ABB RobotStudio station: Inverted.rspag

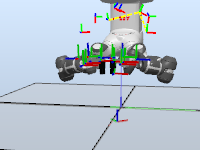
--- station ---
Station DEMO (saved by RobotStudio 20.4.9280.0)
Controller RW6.10.01
  mechanical unit ROB_R: IRB14000_0.5_0.5_R, 6 joints, base frame (0, 0, 820) mm, rotated rx 180 ry 0 rz 0 deg
  mechanical unit ROB_R_7: IRB14000_0.5_0.5_R, 1 joints, base frame (0, 0, 820) mm, rotated rx 180 ry 0 rz 0 deg
  mechanical unit ROB_L: IRB14000_0.5_0.5_L, 6 joints, base frame (0, 0, 820) mm, rotated rx 180 ry 0 rz 0 deg
  mechanical unit ROB_L_7: IRB14000_0.5_0.5_L, 1 joints, base frame (0, 0, 820) mm, rotated rx 180 ry 0 rz 0 deg
Layout (positions relative to the parent item):
  - IRB14000_0.5_0.5 [mechanism, from Robots\IRB14000_0.5_0.5__01.rslib] at (0, 0, 820) mm, rotated rx 180 ry 0 rz 0 deg
  - IRB14000_0.5_0.5_R [mechanism, from Robots\IRB14000_0.5_0.5__01.rslib] at (0, 0, 820) mm, rotated rx 180 ry 0 rz 0 deg; joint values [0.956, -0.6515, -0.6762, 0.5544, 3.1216, 1.0782, 0.2397] (rad or m)
  - IRB14000_0.5_0.5_L [mechanism, from Robots\IRB14000_0.5_0.5__01.rslib] at (0, 0, 820) mm, rotated rx 180 ry 0 rz 0 deg; joint values [-0.9175, -0.6335, 0.6594, 0.5525, 3.1588, 1.0767, -3.4124] (rad or m)
  - cam1 [part] at (530.01, -66.08, 390.5) mm, rotated rx -90 ry 1.82 rz -90 deg
  - cam2 [part] at (530.01, 64.49, 340.52) mm, rotated rx 90 ry 1.82 rz 90 deg
Attachment: cam2 is attached to IRB14000_0.5_0.5_R / Link7
Attachment: cam1 is attached to IRB14000_0.5_0.5_L / Link7
Targets, tools, work objects and paths stored in the station and not in the controller backup, written as RAPID:
! task T_ROB_R
MODULE MainModule
  VAR syncident synco;
  VAR syncident syncon;
  VAR syncident syncoff;
  VAR jointtarget jtraised10:=[[70.951,-118.367,40.9926,106.328,50.1338,-20.9947],[-83.9002,9E+09,9E+09,9E+09,9E+09,9E+09]];
  PROC runexperiment()
    Reset Collision_Avoidance;
    ConfL \Off;
    WaitSyncTask synco,tasklist;
    WaitTime nwaittime;
    WaitSyncTask synco,tasklist;
  ENDPROC
  PROC goto800()
    Reset Collision_Avoidance;
    ConfL \Off;
  ENDPROC
  PROC runallold()
    goto1100;
    goto1400;
    goto1100;
  ENDPROC
  PROC MainOld()
    Reset Collision_Avoidance;
  ENDPROC
  PROC Mainew()
    Reset Collision_Avoidance;
  ENDPROC
ENDMODULE

! task T_ROB_R
MODULE YuMiLib_Params_R
  TASK PERS tooldata tVacuum2:=[TRUE,[[-63.5,18.5,37.5],[0.707106781,0,-0.707106781,0]],[0.28,[7.1,11.9,47.3],[1,0,0,0],0.00025,0.00029,0.00012]];
  TASK PERS tooldata tVacuum1:=[TRUE,[[63.5,18.5,37.5],[0.707106781,0,0.707106781,0]],[0.248,[8.6,11.7,52.7],[1,0,0,0],0.00021,0.00024,0.00009]];
  TASK PERS tooldata tHandCamera:=[TRUE,[[-7.79332,26.2553,35.637],[0.507106,-0.492819,-0.512337,-0.487323]],[0.262,[7.8,11.9,50.7],[1,0,0,0],0.00022,0.00024,0.00009]];
  TASK PERS tooldata tGripper:=[TRUE,[[0,0,136],[1,0,0,0]],[0.23,[8.2,11.7,52],[1,0,0,0],0.00021,0.00024,0.00009]];
  TASK PERS wobjdata WObj_Vision:=[FALSE,TRUE,"",[[401.591,32.4092,0],[0.424655,-0.000000122,-0.000000191,0.905355]],[[0,0,0],[1,0,0,0]]];
  TASK PERS wobjdata WObj_FollowRobL:=[FALSE,FALSE,"ROB_L",[[0,0,0],[1,0,0,0]],[[0,0,0],[1,0,0,0]]];
ENDMODULE

! task T_ROB_R
MODULE YuMiLibExamplesR
  PERS wobjdata TrayWObj:=[FALSE,TRUE,"",[[0,0,0],[1,0,0,0]],[[0,0,0],[1,0,0,0]]];
  PROC YLExample_MoveYSyncProc()
    ConfL \Off;
    ConfL \On;
  ENDPROC
  PROC YLExample_MoveYCollision()
    ConfL \Off;
    ConfL \On;
  ENDPROC
ENDMODULE

! task T_ROB_R
MODULE Data
  TASK PERS tooldata tool1:=[TRUE,[[-49.461,-63.6951,27.321],[1,0,0,0]],[0.23,[-49.461,-63.6951,27.321],[1,0,0,0],0,0,0]];
  PERS tooldata tMarker:=[TRUE,[[0,0,14],[1,0,0,0]],[0.001,[0,0,0.001],[1,0,0,0],0,0,0]];
  TASK PERS tooldata camup:=[TRUE,[[-55.3,0,21.2],[1,0,0,0]],[0.23,[-55.3,0,21.2],[1,0,0,0],0,0,0]];
  PERS wobjdata woupsidedown:=[FALSE,TRUE,"",[[0,0,0],[1,0,0,0]],[[0,0,0],[1,0,0,0]]];
  PERS wobjdata wobj0New:=[FALSE,TRUE,"",[[0,0,0],[0,0,0,1]],[[0,0,0],[1,0,0,0]]];
  TASK PERS wobjdata flangeRobL:=[FALSE,FALSE,"ROB_L",[[0,0,0],[1,0,0,0]],[[0,0,0],[1,0,0,0]]];
  TASK PERS wobjdata flangeRobR:=[FALSE,FALSE,"ROB_R",[[0,0,0],[1,0,0,0]],[[0,0,0],[1,0,0,0]]];
  VAR syncident syncpoint;
  VAR syncident syncraise;
  VAR syncident syncbat1;
  VAR syncident syncbat2;
ENDMODULE

! task T_ROB_L
MODULE MainModule
  VAR syncident syncon;
  VAR syncident syncoff;
  PROC runexperiment()
    Reset Collision_Avoidance;
    ConfL \Off;
    WaitSyncTask synco,tasklist;
    WaitTime nwaittime;
    WaitSyncTask synco,tasklist;
  ENDPROC
  PROC goto800()
    Reset Collision_Avoidance;
    ConfL \Off;
  ENDPROC
  PROC runallold()
    goto1100;
    goto1400;
    goto1100;
  ENDPROC
ENDMODULE

! task T_ROB_L
MODULE YuMiLib_Params_L
  TASK PERS tooldata tVacuum2:=[TRUE,[[-63.5,18.5,37.5],[0.707106781,0,-0.707106781,0]],[0.28,[7.1,11.9,47.3],[1,0,0,0],0.00025,0.00029,0.00012]];
  TASK PERS tooldata tVacuum1:=[TRUE,[[63.5,18.5,37.5],[0.707106781,0,0.707106781,0]],[0.248,[8.6,11.7,52.7],[1,0,0,0],0.00021,0.00024,0.00009]];
  TASK PERS tooldata tHandCamera:=[TRUE,[[-7.79332,26.2553,35.637],[0.507106,-0.492819,-0.512337,-0.487323]],[0.262,[7.8,11.9,50.7],[1,0,0,0],0.00022,0.00024,0.00009]];
  TASK PERS tooldata tGripper:=[TRUE,[[0,0,136],[1,0,0,0]],[0.23,[8.2,11.7,52],[1,0,0,0],0.00021,0.00024,0.00009]];
  TASK PERS wobjdata WObj_Vision:=[FALSE,TRUE,"",[[401.591,32.4092,0],[0.424655,-0.000000122,-0.000000191,0.905355]],[[0,0,0],[1,0,0,0]]];
  TASK PERS wobjdata WObj_FollowRobR:=[FALSE,FALSE,"ROB_R",[[0,0,0],[1,0,0,0]],[[0,0,0],[1,0,0,0]]];
ENDMODULE

! task T_ROB_L
MODULE Data
  PERS tooldata tool1:=[TRUE,[[5.46165,-3.35898,214.586],[1,0,0,0]],[0.23,[0,0,0.001],[1,0,0,0],0,0,0]];
  TASK PERS tooldata camup:=[TRUE,[[55.3,0,21.2],[1,0,0,0]],[0.23,[-55.3,0,21.2],[1,0,0,0],0,0,0]];
  PERS wobjdata woupsidedown:=[FALSE,TRUE,"",[[0,0,-710],[0,0,0,1]],[[0,0,0],[1,0,0,0]]];
  TASK PERS wobjdata flangeRobL:=[FALSE,FALSE,"ROB_L",[[0,0,0],[1,0,0,0]],[[0,0,0],[1,0,0,0]]];
  TASK PERS wobjdata flangeRobR:=[FALSE,FALSE,"ROB_R",[[0,0,0],[1,0,0,0]],[[0,0,0],[1,0,0,0]]];
  PERS wobjdata floor:=[FALSE,TRUE,"",[[0,0,0],[1,0,0,0]],[[0,0,0],[1,0,0,0]]];
  PERS wobjdata basetest:=[FALSE,TRUE,"",[[0,0,410],[0,0,0,1]],[[0,0,0],[1,0,0,0]]];
  VAR syncident synco;
  VAR syncident syncraise;
  VAR syncident syncbat1;
  VAR syncident syncbat2;
  VAR syncident syncpoint;
ENDMODULE

! task T_ROB_L
MODULE YuMiLibExamplesL
  PERS wobjdata TrayWObj:=[FALSE,TRUE,"",[[0,0,0],[1,0,0,0]],[[0,0,0],[1,0,0,0]]];
  PROC YLExample_MoveYSyncProc()
    ConfL \Off;
    ConfL \On;
  ENDPROC
  PROC YLExample_MoveYCollision()
    ConfL \Off;
    ConfL \On;
  ENDPROC
ENDMODULE


--- Backups/RW6.10.01/RAPID/TASK1/PROGMOD/Data.mod ---
MODULE Data

    ! Tooldata for the right camera.
    TASK PERS tooldata tCamR:=[TRUE,[[-55.3,0,21.2],[1,0,0,0]],[0.23,[-55.3,0,21.2],[1,0,0,0],0,0,0]];
    TASK PERS tooldata tCamR_orig:=[TRUE,[[-55.3,0,21.2],[1,0,0,0]],[0.23,[-55.3,0,21.2],[1,0,0,0],0,0,0]];

    TASK PERS robtarget origR := [[456,35,1099.44],[0.507892,0.491981,0.507892,0.491981],[1,2,0,4],[165,9E+9,9E+9,9E+9,9E+9,9E+9]];
    !Additional rotational adjustments

    !Additional rotational adjustments
    VAR num x_offs:=0.0;
    VAR num y_offs:=0;!0.12;
    VAR num z_offs:=0;!-1.00;

    !Data for the experiment
    VAR num distances{20}:=[50,60,70,80,90,100,110,120,130,140,150,160,170,180,190,200,210,220,230,240];
    PERS num nWaittime:=5;
    PERS wobjdata wobjHeart:=[FALSE,TRUE,"",[[0,0,1550],[0,0,1,0]],[[0,0,0],[1,0,0,0]]];
    PERS speeddata speedSlow:=[50,50,5000,5000];
    PERS num nRadius{2}:=[1100, 1400];
    PERS pos convergencePos{2} := [[0, 0, 0], [0, 0, 300]]; !z will be added to this position!

    !Adjusting the x and z position of the convergence points.
    PERS num x:= 456;
    PERS num z:= 1550;



    !For synchronization
    PERS tasks tasklist{2}:=[["T_ROB_R"],["T_ROB_L"]];
    VAR syncident syncpoint;

    !The Stereo2 app reads this status message and displays it on the Flexpendant.
    PERS string myStatus:="Dist 110 h = 1100";


    !For moving into a raised position and to resting aka 'bat' position
    VAR syncident syncraise;
    VAR syncident syncbat1;
    VAR syncident syncbat2;
    VAR jointtarget jtraised:=[[66.0331,-85.1911,41.3253,139.052,44.5799,5.71225],[-62.1903,9E+09,9E+09,9E+09,9E+09,9E+09]];
    VAR jointtarget jtbat:=[[64.6304,-143.384,34.5095,60.7933,53.7269,8.84934],[-140.721,9E+09,9E+09,9E+09,9E+09,9E+09]];
    VAR jointtarget jtraisedVia:=[[70.951,-118.367,40.9926,106.328,50.1338,-20.9947],[-83.9002,9E+09,9E+09,9E+09,9E+09,9E+09]];


ENDMODULE

--- Backups/RW6.10.01/RAPID/TASK1/PROGMOD/MainModule.mod ---
MODULE MainModule




    PROC Main()
        runall;
    ENDPROC

    PROC goToCalibPos()
        VAR jointtarget calibPos := [[-0.00840108,-129.997,30.0284,-0.019315,40.0852,-0.0138285],[-135.001,9E+09,9E+09,9E+09,9E+09,9E+09]];
        MoveAbsJ calibPos\NoEOffs,v1000,z50,tool0;
    ENDPROC

    PROC runall()

        FOR i FROM 1 TO DIM(nRadius, 1) DO
            runtest convergencePos{i}, nRadius{i};
        ENDFOR
    ENDPROC



    PROC MoveToDist(num dist,num h\speeddata sp, PERS wobjdata wobjHeart)
        VAR robtarget position:=[[365,-10,1000],[0.5,0.5,0.5,0.5],[1,-2,-2,4],[165,9E+09,9E+09,9E+09,9E+09,9E+09]];
        VAR num angle;
        VAR num halfdist;
        VAR num rads;
        VAR num zh;
        VAR num y;
        VAR speeddata speed;


        halfdist:=dist/2;
        speed:=speedSlow;
        angle:=ASin(halfdist/h);
        y:=h*sin(angle);
        zh:=h*cos(angle);

        position.trans:=[x,y,zh];
        IF Present(sp) THEN
            speed:=sp;
        ENDIF

        MoveL RelTool(position,0,0,0\Rx:=x_offs\Ry:=y_offs\Rz:=-(angle+z_offs)),speed,fine,tCamR\WObj:=wobjHeart;

    ENDPROC


    PROC inc()
        VAR num s:=1;
        z := z + s;
        goto1100;
    ENDPROC


    PROC incinc()

        VAR num s:=5;
        z := z + s;
        goto1100;
    ENDPROC


    PROC dec()

        VAR num s:=-1;
        z := z + s;
        goto1100;
    ENDPROC


    PROC decdec()
        VAR num s:=-5;
        z := z + s;
        goto1100;
    ENDPROC

    PROC incX()
        VAR num s:=1;
        x:=x+s;
        goto1100;
    ENDPROC


    PROC incincX()

        VAR num s:=5;
        x:=x+s;
        goto1100;
    ENDPROC


    PROC decX()

        VAR num s:=-1;
        x:=x+s;
        goto1100;
    ENDPROC


    PROC decdecX()

        VAR num s:=-5;
        x:=x+s;
        goto1100;
    ENDPROC

    PROC gotoX1()
        ReSet Collision_Avoidance;
        ConfL\Off;
        wobjHeart.uframe.trans := [convergencePos{1}.x, convergencePos{1}.y, convergencePos{1}.z + z];
        WaitSyncTask syncpoint,tasklist;
        !origR := CRobT(\Tool:=tCamR_orig);
        MoveToDist distances{3},nRadius{1}\sp:=v100, wobjHeart;
    ENDPROC

    PROC L_update()

    ENDPROC


    PROC R_update()
        VAR robtarget new;
        VAR pose orig_pose;
        VAR pose new_pose;
        VAR pose diff;
        VAR pose tool_pose;
        VAR btnres answer;
        tool_pose := tCamR_orig.tframe;
        new := CRobT(\Tool:=tCamR_orig);
        orig_pose := [origR.trans, origR.rot];
        new_pose := [new.trans, new.rot];
        diff := PoseMult(PoseInv(new_pose), orig_pose);
        tCamR.tframe := PoseMult(tool_pose, diff);


    ENDPROC

    PROC reset_tool()
        tCamR := tCamR_orig;

    ENDPROC

    PROC gotoX2()

        ReSet Collision_Avoidance;
        ConfL\Off;
        wobjHeart.uframe.trans := [convergencePos{1}.x, convergencePos{1}.y, convergencePos{1}.z+z];
        WaitSyncTask syncpoint,tasklist;
        MoveToDist distances{15},nRadius{1}\sp:=v100, wobjHeart;

    ENDPROC


    PROC gofrombatpos()

        ReSet Collision_Avoidance;
        ConfL\Off;
        MoveAbsJ jtraisedVia\NoEOffs,v100,fine,tCamR;
        MoveAbsJ jtraised\NoEOffs,v100,fine,tCamR;
        WaitSyncTask syncraise,tasklist;
    ENDPROC

    PROC gotoraisedpos()
        ReSet Collision_Avoidance;
        ConfL\Off;
        MoveAbsJ jtraised\NoEOffs,v100,fine,tCamR;
        WaitSyncTask syncraise,tasklist;

    ENDPROC

    PROC gotobatpos()
        ReSet Collision_Avoidance;
        ConfL\Off;
        MoveAbsJ jtraised\NoEOffs,v100,fine,tCamR\WObj:=wobjHeart;
        WaitSyncTask syncbat1,tasklist;
        WaitSyncTask syncbat2,tasklist;
        MoveAbsJ jtraisedVia\NoEOffs,v100,fine,tCamR;
        MoveAbsJ jtbat\NoEOffs,v100,fine,tCamR;

    ENDPROC



    PROC goto1100()
        ReSet Collision_Avoidance;
        ConfL\Off;
        wobjHeart.uframe.trans := [convergencePos{1}.x, convergencePos{1}.y, convergencePos{1}.z + z];
        WaitSyncTask syncpoint,tasklist;
        MoveToDist distances{1},nRadius{1}\sp:=v100, wobjHeart;
    ENDPROC


    PROC goto1400()
        ReSet Collision_Avoidance;
        ConfL\Off;
        wobjHeart.uframe.trans := [convergencePos{2}.x, convergencePos{2}.y, convergencePos{2}.z + z];
        WaitSyncTask syncpoint,tasklist;
        MoveToDist distances{1},nRadius{2}\sp:=v100, wobjHeart;

    ENDPROC


    PROC run1100()
        runtest convergencePos{1},nRadius{1};
    ENDPROC

    PROC run1400()

        runtest convergencePos{2},nRadius{2};
    ENDPROC



    PROC runtest(pos position,num h)

        ConfL\Off;
        wobjHeart.uframe.trans:=[position.x, position.y, position.z + z];
        WaitSyncTask syncpoint,tasklist;
        ReSet Collision_Avoidance;
        MoveToDist distances{1},h\sp:=v100, wobjHeart;

        FOR i FROM 1 TO Dim(distances,1) DO

            WaitSyncTask syncpoint,tasklist;
            myStatus:="Dist "+NumToStr(distances{i},0)+" h = "+NumToStr(h,0);
            ErrWrite\I,"Started moving. Dist "+NumToStr(distances{i},0)+" h = "+NumToStr(h,0),"";
            MoveToDist distances{i},h, wobjHeart;
            WaitTime nwaittime;
        ENDFOR
        WaitSyncTask syncpoint,tasklist;
    ENDPROC


ENDMODULE

--- Backups/RW6.10.01/RAPID/TASK2/PROGMOD/Data.mod ---
    MODULE Data


    ! Tooldata for the left camera.
    TASK PERS tooldata tCamL:=[TRUE,[[55.3,0,21.2],[1,0,0,0]],[0.23,[55.3,0,21.2],[1,0,0,0],0,0,0]];
    TASK PERS tooldata tCamL_orig:=[TRUE,[[55.3,0,21.2],[1,0,0,0]],[0.23,[55.3,0,21.2],[1,0,0,0],0,0,0]];

    TASK PERS robtarget origL := [[456,-35,1099.44],[0.491981,0.507892,0.491981,0.507892],[-1,2,-2,4],[-163.142,9E+9,9E+9,9E+9,9E+9,9E+9]];

   ! Additional rotational adjustments.
    VAR num x_offs:= 0.0;
    VAR num y_offs:= 0.0;
    VAR num z_offs:=0;!0.43;


    !Data for the experiment. These are shared with the right task and assigned in T_ROB_R/Data
    VAR num distances{20}:=[50,60,70,80,90,100,110,120,130,140,150,160,170,180,190,200,210,220,230,240];
    PERS num nWaittime;
    PERS wobjdata wobjHeart;
    PERS speeddata speedSlow;
    PERS num nRadius{2};
    PERS pos convergencePos{2};


    !Adjusting the x and z position of the convergence points.
    PERS num x;
    PERS num z;



    !For synchronization
    PERS tasks tasklist{2}:=[["T_ROB_R"],["T_ROB_L"]];
    VAR syncident syncpoint;

    !For moving into a raised position and to resting aka 'bat' position
    VAR jointtarget jtraised:=[[-74.7004,-91.3236,43.3868,218.306,45.6835,-171.438],[61.909,9E+09,9E+09,9E+09,9E+09,9E+09]];
    VAR syncident syncraise;
    VAR syncident syncbat1;
    VAR syncident syncbat2;
    VAR jointtarget jtbat:=[[-56.5752,-119.517,21.4015,271.499,49.3732,-213.567],[155.307,9E+09,9E+09,9E+09,9E+09,9E+09]];

ENDMODULE

--- Backups/RW6.10.01/RAPID/TASK2/PROGMOD/MainModule.mod ---
    MODULE MainModule



    PROC goToCalibPos()
        VAR jointtarget calibPos := [[0.00341333,-129.995,30.0196,-0.000788279,40.0913,-0.461743],[134.997,9E+09,9E+09,9E+09,9E+09,9E+09]];
        MoveAbsJ calibPos\NoEOffs,v1000,z50,tool0;
    ENDPROC

    PROC Main()

        runall;
    ENDPROC

    PROC runall()
        FOR i FROM 1 TO DIM(nRadius, 1) DO
            runtest convergencePos{i}, nRadius{i};
        ENDFOR
    ENDPROC



    PROC MoveToDist(num dist,num h,\speeddata sp, PERS wobjdata wobjHeart)
        !   VAR robtarget position := [[0,0,0],[0.0,0.0,0.7071,-0.7071],[1,1,0,4],[143.284,9E+09,9E+09,9E+09,9E+09,9E+09]];
        VAR robtarget position:=[[0,0,0],[0.5,0.5,0.5,0.5],[1,-2,0,0],[-163.142,9E+09,9E+09,9E+09,9E+09,9E+09]];
        VAR num angle;
        VAR num halfdist;
        VAR num rads;
        VAR num zh;
        VAR num y;
        VAR speeddata speed;

        halfdist:=dist/2;
        speed:=speedSlow;
        angle:=ASin(halfdist/h);
        y:=h*sin(angle);
        zh:=h*cos(angle);

        position.trans:=[x,-y,zh];
        IF Present(sp) THEN
            speed:=sp;
        ENDIF
        MoveL RelTool(position,0,0,0\Ry:=y_offs\Rz:=angle+z_offs),speed,fine,tCamL\WObj:=wobjHeart;


    ENDPROC





    PROC gotoraisedpos()

        ReSet Collision_Avoidance;
        ConfL\Off;
        WaitSyncTask syncraise,tasklist;
        MoveAbsJ jtraised\NoEOffs,v100,fine,tCamL;

    ENDPROC

    PROC inc()
        goto1100;
    ENDPROC


    PROC incinc()
        goto1100;
    ENDPROC


    PROC dec()
        goto1100;
    ENDPROC


    PROC decdec()
        goto1100;
    ENDPROC



    PROC incX()
        goto1100;
    ENDPROC


    PROC incincX()

        goto1100;
    ENDPROC


    PROC decX()

        goto1100;

    ENDPROC


    PROC decdecX()
        goto1100;

    ENDPROC

    PROC gofrombatpos()
        VAR jointtarget jtVia := [[-68.4054,-105.589,37.6928,245.742,40.601,-189.436],[135.726,9E+09,9E+09,9E+09,9E+09,9E+09]];
        ReSet Collision_Avoidance;
        ConfL\Off;
        WaitSyncTask syncraise,tasklist;
        MoveAbsJ jtVia\NoEOffs,v100,fine,tCamL;
        MoveAbsJ jtraised\NoEOffs,v100,fine,tCamL;

    ENDPROC

    PROC gotobatpos()
        VAR jointtarget jtBatPos := [[-68.4054,-105.589,37.6928,245.742,40.601,-189.436],[135.726,9E+09,9E+09,9E+09,9E+09,9E+09]];
        ReSet Collision_Avoidance;
        ConfL\Off;
        MoveAbsJ jtraised\NoEOffs,v100,fine,tCamL;
        WaitSyncTask syncbat1,tasklist;
        MoveAbsJ jtBatPos\NoEOffs,v100,fine,tCamL;
        MoveAbsJ jtbat\NoEOffs,v100,fine,tCamL;
        WaitSyncTask syncbat2,tasklist;
    ENDPROC


    PROC gotoX1()

        ReSet Collision_Avoidance;
        ConfL\Off;
        WaitSyncTask syncpoint,tasklist;
        !origL := CRobT(\Tool:=tCamL_orig);

        MoveToDist distances{3},nRadius{1}\sp:=v100, wobjHeart;
    ENDPROC


    PROC L_update()
        VAR robtarget new;
        VAR pose orig_pose;
        VAR pose new_pose;
        VAR pose diff;
        VAR pose tool_pose;
        VAR btnres answer;
        tool_pose := tCamL_orig.tframe;
        new := CRobT(\Tool:=tCamL_orig);
        orig_pose := [origL.trans, origL.rot];
        new_pose := [new.trans, new.rot];
        diff := PoseMult(PoseInv(new_pose), orig_pose);
        tCamL.tframe := PoseMult(tool_pose, diff);


    ENDPROC


    PROC R_update()
    ENDPROC

    PROC reset_tool()
        tCamL := tCamL_orig;

    ENDPROC

    PROC gotoX2()
        ReSet Collision_Avoidance;
        ConfL\Off;
        WaitSyncTask syncpoint,tasklist;
        MoveToDist distances{15},nRadius{1}\sp:=v100, wobjHeart;

    ENDPROC


    PROC goto1100()
        ReSet Collision_Avoidance;
        ConfL\Off;
        WaitSyncTask syncpoint,tasklist;
        MoveToDist distances{1},nRadius{1}\sp:=v100, wobjHeart;

    ENDPROC




    PROC goto1400()
        ReSet Collision_Avoidance;
        ConfL\Off;
        WaitSyncTask syncpoint,tasklist;
        MoveToDist distances{1},nRadius{2}\sp:=v100, wobjHeart;

    ENDPROC


    PROC run1100()
        runtest convergencePos{1},nRadius{1};
    ENDPROC

    PROC run1400()

        runtest convergencePos{2},nRadius{2};
    ENDPROC



    PROC runtest(pos position,num h)
        ReSet Collision_Avoidance;
        ConfL\Off;
        WaitSyncTask syncpoint,tasklist;

        MoveToDist distances{1},h\sp:=v100, wobjHeart;

        FOR i FROM 1 TO Dim(distances,1) DO
            WaitSyncTask syncpoint,tasklist;
            MoveToDist distances{i},h, wobjHeart;
            WaitTime nwaittime;
        ENDFOR

        WaitSyncTask syncpoint,tasklist;
    ENDPROC

ENDMODULE

--- Backups/RW6.10.01/SYSPAR/EIO.cfg ---
EIO:CFG_1.0:6:1::
#
SYSSIG_IN:

      -Signal "Collision_Avoidance" -Action "CollAvoidance"
#
INDUSTRIAL_NETWORK:

      -Name "DeviceNet" -Label "DeviceNet Master/Slave Network" -Address "2"
#
EIO_CROSS:

      -Name "Cross_Signal_Lamp" -Res "Signal_Lamp" -Act1 "DRV1BRAKE"
#
EIO_SIGNAL_SAFELEVEL:

      -Name "FlangePowerSafeLevel" -ActionWhenStartup "Last"

      -Name "SGcmdSafeLevel" -ActionWhenAccessible "Default"
#
ETHERNETIP_DEVICE:

      -Name "Hand_R" -StateWhenStartup "Deactivated" -VendorName "ABB"\
      -ProductName "EtherNet/IP EIP" -Label "2" -Address "192.168.125.30"\
      -VendorId 75 -ProductCode 1 -OutputAssembly 100 -InputAssembly 101\
      -InputConnectionType "POINT2POINT" -OutputSize 10 -InputSize 10\
      -O2T_RPI 10000 -T2O_RPI 10000 -ConnectionTimeoutMultiplier 2

      -Name "Hand_L" -StateWhenStartup "Deactivated" -VendorName "ABB"\
      -ProductName "EtherNet/IP EIP" -Label "1" -Address "192.168.125.40"\
      -VendorId 75 -ProductCode 1 -OutputAssembly 100 -InputAssembly 101\
      -InputConnectionType "POINT2POINT" -OutputSize 10 -InputSize 10\
      -O2T_RPI 10000 -T2O_RPI 10000 -ConnectionTimeoutMultiplier 2
#
DEVICENET_DEVICE:

      -Name "D652_10" -VendorName "ABB Robotics" -ProductName "24 VDC Unit"\
      -Address 10 -ProductCode 26 -DeviceType 7 -ConnectionType "COS"\
      -OutputSize 2 -InputSize 2
#
DEVICENET_INTERNAL_DEVICE:

      -Name "DN_Internal_Device" -VendorName "ABB Robotics"\
      -ProductName "DeviceNet Internal Slave Device"
#
EIO_SIGNAL:

      -Name "custom_DI_0" -SignalType "DI" -Device "D652_10" -DeviceMap "0"

      -Name "custom_DI_1" -SignalType "DI" -Device "D652_10" -DeviceMap "1"

      -Name "custom_DI_2" -SignalType "DI" -Device "D652_10" -DeviceMap "2"

      -Name "custom_DI_3" -SignalType "DI" -Device "D652_10" -DeviceMap "3"

      -Name "custom_DI_4" -SignalType "DI" -Device "D652_10" -DeviceMap "4"

      -Name "custom_DI_5" -SignalType "DI" -Device "D652_10" -DeviceMap "5"

      -Name "custom_DI_6" -SignalType "DI" -Device "D652_10" -DeviceMap "6"

      -Name "custom_DI_7" -SignalType "DI" -Device "D652_10" -DeviceMap "7"

      -Name "custom_DO_0" -SignalType "DO" -Device "D652_10" -DeviceMap "0"

      -Name "custom_DO_1" -SignalType "DO" -Device "D652_10" -DeviceMap "1"

      -Name "custom_DO_2" -SignalType "DO" -Device "D652_10" -DeviceMap "2"

      -Name "custom_DO_3" -SignalType "DO" -Device "D652_10" -DeviceMap "3"

      -Name "custom_DO_4" -SignalType "DO" -Device "D652_10" -DeviceMap "4"

      -Name "custom_DO_5" -SignalType "DO" -Device "D652_10" -DeviceMap "5"

      -Name "custom_DO_6" -SignalType "DO" -Device "D652_10" -DeviceMap "6"

      -Name "custom_DO_7" -SignalType "DO" -Device "D652_10" -DeviceMap "7"

      -Name "hall_sensor_joint_1" -SignalType "DI" -Device "D652_10"\
      -DeviceMap "8"

      -Name "hall_sensor_joint_2" -SignalType "DI" -Device "D652_10"\
      -DeviceMap "9"

      -Name "hall_sensor_joint_3" -SignalType "DI" -Device "D652_10"\
      -DeviceMap "11"

      -Name "hall_sensor_joint_4" -SignalType "DI" -Device "D652_10"\
      -DeviceMap "12"

      -Name "hall_sensor_joint_5" -SignalType "DI" -Device "D652_10"\
      -DeviceMap "13"

      -Name "hall_sensor_joint_6" -SignalType "DI" -Device "D652_10"\
      -DeviceMap "14"

      -Name "hall_sensor_joint_7" -SignalType "DI" -Device "D652_10"\
      -DeviceMap "10"

      -Name "hall_sensor_24V_ROB_R" -SignalType "DO" -Device "D652_10"\
      -DeviceMap "8"

      -Name "hall_sensor_24V_ROB_L" -SignalType "DO" -Device "D652_10"\
      -DeviceMap "9"

      -Name "flange_24V_ROB_R" -SignalType "DO" -Device "D652_10"\
      -DeviceMap "10" -SafeLevel "FlangePowerSafeLevel"

      -Name "flange_24V_ROB_L" -SignalType "DO" -Device "D652_10"\
      -DeviceMap "11" -SafeLevel "FlangePowerSafeLevel"

      -Name "Signal_Lamp" -SignalType "DO" -Device "D652_10" -DeviceMap "12"

      -Name "Collision_Avoidance" -SignalType "DO" -Access "All" -Default 1

      -Name "hand_CmdGripper_R" -SignalType "GO" -Device "Hand_R"\
      -Label "Hand Command Right" -DeviceMap "0-4" -Category "HandRight"\
      -Access "All" -SafeLevel "SGcmdSafeLevel"

      -Name "hand_CmdClearErr_R" -SignalType "DO" -Device "Hand_R"\
      -Label "Clear Error Right" -DeviceMap "7" -Category "HandRight"\
      -Access "All"

      -Name "hand_MaxPosition_R" -SignalType "GO" -Device "Hand_R"\
      -Label "Max Position Right" -DeviceMap "8-15" -Category "HandRight"\
      -Access "All" -Default 100

      -Name "hand_MinPosition_R" -SignalType "GO" -Device "Hand_R"\
      -Label "Min Position Right" -DeviceMap "16-23" -Category "HandRight"\
      -Access "All" -Default 50

      -Name "hand_MaxSpeed_R" -SignalType "GO" -Device "Hand_R"\
      -Label "Max Speed Right" -DeviceMap "24-31" -Category "HandRight"\
      -Access "All" -Default 200

      -Name "hand_HoldForce_R" -SignalType "GO" -Device "Hand_R"\
      -Label "Hold Force Right" -DeviceMap "40-47" -Category "HandRight"\
      -Access "All" -Default 120

      -Name "hand_CmdVacuum1_R" -SignalType "DO" -Device "Hand_R"\
      -Label "Vacuum 1 Right" -DeviceMap "48" -Category "HandRight"\
      -Access "All"

      -Name "hand_CmdVacuum2_R" -SignalType "DO" -Device "Hand_R"\
      -Label "Vacuum 2 Right" -DeviceMap "49" -Category "HandRight"\
      -Access "All"

      -Name "hand_CmdBlowoff1_R" -SignalType "DO" -Device "Hand_R"\
      -Label "BlowOff 1 Right" -DeviceMap "50" -Category "HandRight"\
      -Access "All"

      -Name "hand_CmdBlowoff2_R" -SignalType "DO" -Device "Hand_R"\
      -Label "BlowOff 2 Right" -DeviceMap "51" -Category "HandRight"\
      -Access "All"

      -Name "hand_SysState_R" -SignalType "GI" -Device "Hand_R"\
      -Label "Finger State Right" -DeviceMap "0-4" -Category "HandRight"\
      -Access "All"

      -Name "hand_SysError_R" -SignalType "GI" -Device "Hand_R"\
      -Label "Finger Error Right" -DeviceMap "32-39" -Category "HandRight"\
      -Access "All"

      -Name "hand_StatusCalibrated_R" -SignalType "DI" -Device "Hand_R"\
      -Label "Calibrated Right" -DeviceMap "5" -Category "HandRight"\
      -Access "All"

      -Name "hand_ActualPosition_R" -SignalType "GI" -Device "Hand_R"\
      -Label "Actual Position Right" -DeviceMap "8-15" -Category "HandRight"\
      -Access "All"

      -Name "hand_ActualSpeed_R" -SignalType "GI" -Device "Hand_R"\
      -Label "Actual Speed Right" -DeviceMap "16-23" -Category "HandRight"\
      -Access "All"

      -Name "hand_StatusCamLinked_R" -SignalType "DI" -Device "Hand_R"\
      -Label "Camera Connection Right" -DeviceMap "40" -Category "HandRight"\
      -Access "All"

      -Name "hand_SoftwareVersion_R" -SignalType "GI" -Device "Hand_R"\
      -Label "Software Version Right" -DeviceMap "41-47" -Category "HandRight"\
      -Access "All"

      -Name "hand_StatusVacuum1_R" -SignalType "DI" -Device "Hand_R"\
      -Label "Vacuum 1 Right Status" -DeviceMap "48" -Category "HandRight"\
      -Access "All"

      -Name "hand_StatusVacuum2_R" -SignalType "DI" -Device "Hand_R"\
      -Label "Vacuum 1 Right Status" -DeviceMap "49" -Category "HandRight"\
      -Access "All"

      -Name "hand_StatusBlowoff1_R" -SignalType "DI" -Device "Hand_R"\
      -Label "SuncTool 1 Right Status" -DeviceMap "50" -Category "HandRight"\
      -Access "All"

      -Name "hand_StatusBlowoff2_R" -SignalType "DI" -Device "Hand_R"\
      -Label "SuncTool 1 Right Status" -DeviceMap "51" -Category "HandRight"\
      -Access "All"

      -Name "hand_ActualPressure1_R" -SignalType "GI" -Device "Hand_R"\
      -Label "Vacuum pressure1 Right" -DeviceMap "64-71" -Category "HandRight"\
      -Access "All"

      -Name "hand_ActualPressure2_R" -SignalType "GI" -Device "Hand_R"\
      -Label "Vacuum pressure2 Right" -DeviceMap "72-79" -Category "HandRight"\
      -Access "All"

      -Name "hand_SecurityKey_R" -SignalType "GO" -Device "Hand_R"\
      -Label "Security key right" -DeviceMap "64-71" -Category "HandRight"\
      -Access "All"

      -Name "hand_TftPFtpMode_R" -SignalType "DI" -Device "Hand_R"\
      -Label "Hand firmware update mode" -DeviceMap "7" -Category "HandRight"\
      -Access "All"

      -Name "hand_CmdGripper_L" -SignalType "GO" -Device "Hand_L"\
      -Label "Hand Command Left" -DeviceMap "0-4" -Category "HandLeft"\
      -Access "All" -SafeLevel "SGcmdSafeLevel"

      -Name "hand_CmdClearErr_L" -SignalType "DO" -Device "Hand_L"\
      -Label "Clear Error Left" -DeviceMap "7" -Category "HandLeft"\
      -Access "All"

      -Name "hand_MaxPosition_L" -SignalType "GO" -Device "Hand_L"\
      -Label "Max Position Left" -DeviceMap "8-15" -Category "HandLeft"\
      -Access "All" -Default 100

      -Name "hand_MinPosition_L" -SignalType "GO" -Device "Hand_L"\
      -Label "Min Position Left" -DeviceMap "16-23" -Category "HandLeft"\
      -Access "All" -Default 50

      -Name "hand_MaxSpeed_L" -SignalType "GO" -Device "Hand_L"\
      -Label "Max Speed Left" -DeviceMap "24-31" -Category "HandLeft"\
      -Access "All" -Default 200

      -Name "hand_HoldForce_L" -SignalType "GO" -Device "Hand_L"\
      -Label "Hold Force Left" -DeviceMap "40-47" -Category "HandLeft"\
      -Access "All" -Default 120

      -Name "hand_CmdVacuum1_L" -SignalType "DO" -Device "Hand_L"\
      -Label "Vacuum 1 Left" -DeviceMap "48" -Category "HandLeft" -Access "All"

      -Name "hand_CmdVacuum2_L" -SignalType "DO" -Device "Hand_L"\
      -Label "Vacuum 2 Left" -DeviceMap "49" -Category "HandLeft" -Access "All"

      -Name "hand_CmdBlowoff1_L" -SignalType "DO" -Device "Hand_L"\
      -Label "BlowOff 1 Left" -DeviceMap "50" -Category "HandLeft" -Access "All"

      -Name "hand_CmdBlowoff2_L" -SignalType "DO" -Device "Hand_L"\
      -Label "BlowOff 2 Left" -DeviceMap "51" -Category "HandLeft" -Access "All"

      -Name "hand_SysState_L" -SignalType "GI" -Device "Hand_L"\
      -Label "Finger State Left" -DeviceMap "0-4" -Category "HandLeft"\
      -Access "All"

      -Name "hand_SysError_L" -SignalType "GI" -Device "Hand_L"\
      -Label "Finger Error Left" -DeviceMap "32-39" -Category "HandLeft"\
      -Access "All"

      -Name "hand_StatusCalibrated_L" -SignalType "DI" -Device "Hand_L"\
      -Label "Calibrated Left" -DeviceMap "5" -Category "HandLeft" -Access "All"

      -Name "hand_ActualPosition_L" -SignalType "GI" -Device "Hand_L"\
      -Label "Actual Position Left" -DeviceMap "8-15" -Category "HandLeft"\
      -Access "All"

      -Name "hand_ActualSpeed_L" -SignalType "GI" -Device "Hand_L"\
      -Label "Actual Speed Left" -DeviceMap "16-23" -Category "HandLeft"\
      -Access "All"

      -Name "hand_StatusCamLinked_L" -SignalType "DI" -Device "Hand_L"\
      -Label "Camera Connection Left" -DeviceMap "40" -Category "HandLeft"\
      -Access "All"

      -Name "hand_SoftwareVersion_L" -SignalType "GI" -Device "Hand_L"\
      -Label "Software Version Left" -DeviceMap "41-47" -Category "HandLeft"\
      -Access "All"

      -Name "hand_StatusVacuum1_L" -SignalType "DI" -Device "Hand_L"\
      -Label "Vacuum 1 Left Status" -DeviceMap "48" -Category "HandLeft"\
      -Access "All"

      -Name "hand_StatusVacuum2_L" -SignalType "DI" -Device "Hand_L"\
      -Label "Vacuum 1 Left Status" -DeviceMap "49" -Category "HandLeft"\
      -Access "All"

      -Name "hand_StatusBlowoff1_L" -SignalType "DI" -Device "Hand_L"\
      -Label "SuncTool 1 Left Status" -DeviceMap "50" -Category "HandLeft"\
      -Access "All"

      -Name "hand_StatusBlowoff2_L" -SignalType "DI" -Device "Hand_L"\
      -Label "SuncTool 1 Left Status" -DeviceMap "51" -Category "HandLeft"\
      -Access "All"

      -Name "hand_ActualPressure1_L" -SignalType "GI" -Device "Hand_L"\
      -Label "Vacuum pressure1 Left" -DeviceMap "64-71" -Category "HandLeft"\
      -Access "All"

      -Name "hand_ActualPressure2_L" -SignalType "GI" -Device "Hand_L"\
      -Label "Vacuum pressure2 Left" -DeviceMap "72-79" -Category "HandLeft"\
      -Access "All"

      -Name "hand_SecurityKey_L" -SignalType "GO" -Device "Hand_L"\
      -Label "Security key Left" -DeviceMap "64-71" -Category "HandLeft"\
      -Access "All"

      -Name "hand_TftPFtpMode_L" -SignalType "DI" -Device "Hand_L"\
      -Label "Hand firmware update mode" -DeviceMap "7" -Category "HandLeft"\
      -Access "All"
